INTERFACE INTERNAL I_TagOwner

END_INTERFACE

(* stored: Version 1.1.0.1
   Itf I_TagOwner: Id {75009c1b-4b32-4472-82ce-f26080344dc4} *)
